% RSLogix 500 project Tarea_4_semaforo_limites_logix_500.RSS, saved by version 8.30.00.16 %
PROJECT "UNTITLED"    % processor: MicroLogix 1000 %

PROGRAM FILES
  LAD 2 "MAIN_PROG"  10 rungs
  LAD 3 "USER_FAULT"  1 rungs
  LAD 4 "HSC_INT"  1 rungs
  LAD 5 "STI_INT"  1 rungs
  LAD 6, 7, 8, 9, 10, 11, 12, 13, 14, 15, 16: only END

DATA FILES
  O0 OUTPUT  1 elements
  I1 INPUT  2 elements
  S2 STATUS  33 elements
  B3 BINARY  32 elements
  T4 TIMER  40 elements
  C5 COUNTER  32 elements
  R6 CONTROL  16 elements
  N7 INTEGER  105 elements

LADDER 2 "MAIN_PROG"
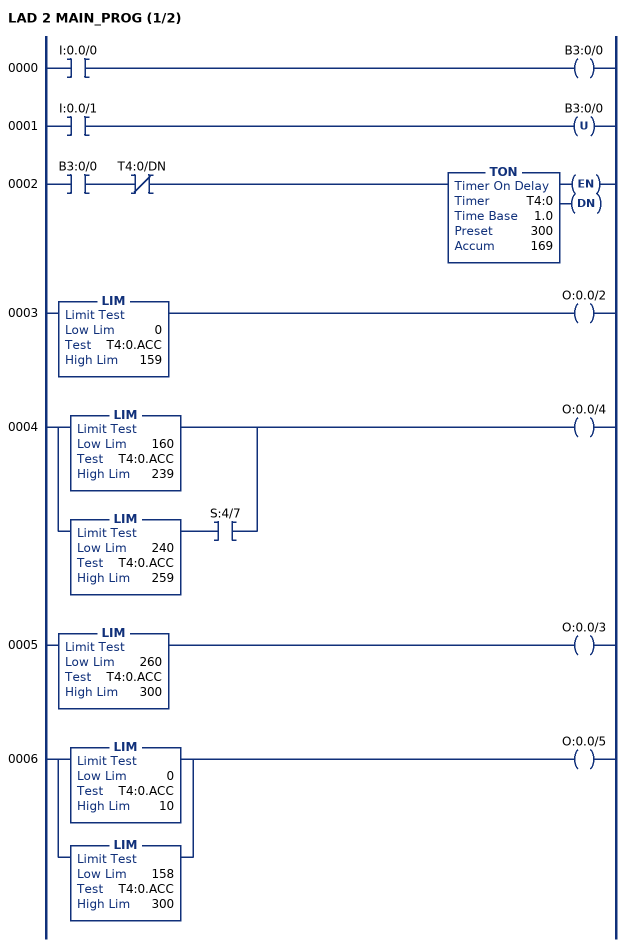
% Rung: 0 %
SOR XIC I:0.0/0 OTE B3:0/0 EOR
% Rung: 1 %
SOR XIC I:0.0/1 OTU B3:0/0 EOR
% Rung: 2 %
SOR XIC B3:0/0 XIO T4:0/DN TON T4:0 1.0 300 169 EOR
% Rung: 3 %
SOR LIM 0 T4:0.ACC 159 OTE O:0.0/2 EOR
% Rung: 4 %
SOR BST LIM 160 T4:0.ACC 239 NXB LIM 240 T4:0.ACC 259 XIC S:4/7 BND OTE O:0.0/4 EOR
% Rung: 5 %
SOR LIM 260 T4:0.ACC 300 OTE O:0.0/3 EOR
% Rung: 6 %
SOR BST LIM 0 T4:0.ACC 10 NXB LIM 158 T4:0.ACC 300 BND OTE O:0.0/5 EOR

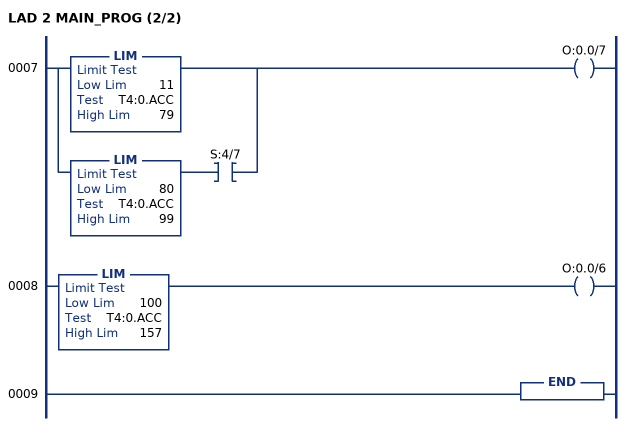
% Rung: 7 %
SOR BST LIM 11 T4:0.ACC 79 NXB LIM 80 T4:0.ACC 99 XIC S:4/7 BND OTE O:0.0/7 EOR
% Rung: 8 %
SOR LIM 100 T4:0.ACC 157 OTE O:0.0/6 EOR
% Rung: 9 %
SOR END EOR

OTHER DOCUMENTED ADDRESSES
  I:1.0/0  START  "I:1/0"

DATA TABLE (non-zero values as saved)
DATA B3
% B3:0 % 0X0001 0X0000 0X0000 0X0000 0X0000 0X0000 0X0000 0X0000 0X0000 0X0000
DATA T4
% .PRE .ACC %
% T4:0 % 300 169
